// Mitsubishi GX Works2 project: IELET2103_Oving2   PLC: FX2N/FX2NC
// IELET2103_Oving2

// global labels: Global1
VAR_GLOBAL
  Nødstoppbryter : BOOL;
  Drasnor_inne : BOOL;
  Drasnor_ute : BOOL;
  Giver_for_port_oppe : BOOL;
  Giver_for_port_nede : BOOL;
  Kontaktor_for_opprulling : BOOL;
  Kontaktor_for_nedrrulling : BOOL;
  Lampe : BOOL;
END_VAR

// task Task_01 (event TRUE, interval 0, priority 31): Oppgave3

PROGRAM Oppgave1a)ST
VAR
  tmp1 : BOOL;
END_VAR
tmp1	:=	 X0 OR (NOT X1 AND M0) AND (M0<>X0) OR NOT M1;

M0 := tmp1; 
M1 :=	tmp1 AND X1;
END_PROGRAM

PROGRAM Oppgave1a)IL
// body in language c0 not rendered
END_PROGRAM

PROGRAM Oppgave1a)LD
(* structured ladder/FBD written out as ST: instructions are called as NAME(EN, inputs, outputs); _pN, _eN, _tN stand for wires *)
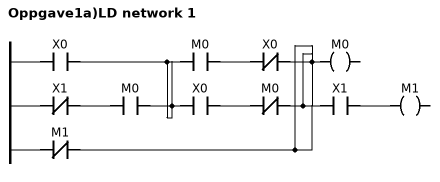
(* network 1 *)
_p1 := X0 OR (NOT X1 AND M0);
_p2 := (_p1 AND M0 AND NOT X0) OR (_p1 AND X0 AND NOT M0) OR (NOT M1);
M0 := _p2;
M1 := _p2 AND X1;
END_PROGRAM

PROGRAM Oppgave1b)LD
(* structured ladder/FBD written out as ST: instructions are called as NAME(EN, inputs, outputs); _pN, _eN, _tN stand for wires *)
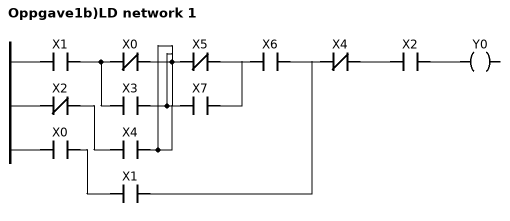
(* network 1 *)
_p1 := (X1 AND NOT X0) OR (X1 AND X3) OR (NOT X2 AND X4);
Y0 := (((((_p1 AND NOT X5) OR (_p1 AND X7)) AND X6) OR (X0 AND X1)) AND NOT X4) AND X2;
END_PROGRAM

PROGRAM Oppgave1b)ST
VAR
  block1 : BOOL;
  block2 : BOOL;
  block3 : BOOL;
  block4 : BOOL;
END_VAR
(*Oppgave 1b) ST*)

block1 := X1 AND (NOT X0 OR X3);
block2 := NOT X2 AND X4;
block3 := (block1 OR block2) AND (NOT X5 OR X7) AND X6;
block4 := block3 OR (X0 AND X1)
 
Y0 := block4 AND NOT X4 AND X2;
END_PROGRAM

PROGRAM Oppgave1c)
(* structured ladder/FBD written out as ST: instructions are called as NAME(EN, inputs, outputs); _pN, _eN, _tN stand for wires *)
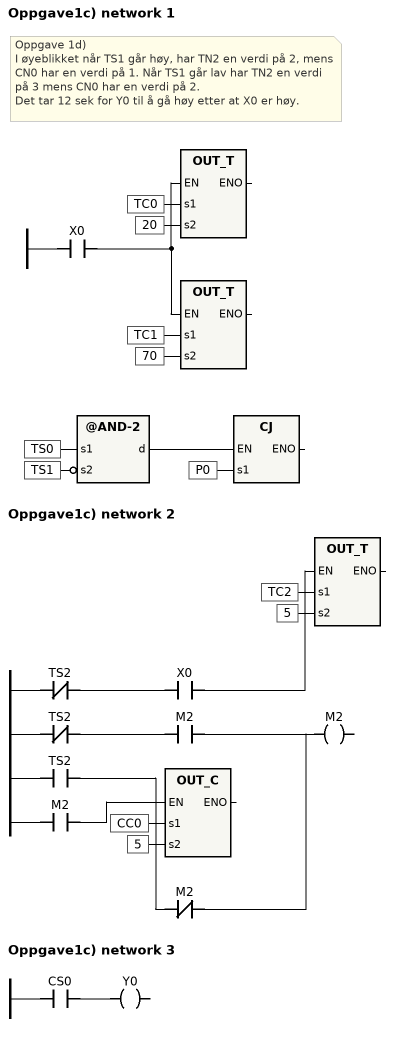
(* network 1 *)
(* Oppgave 1d)  / I øyeblikket når TS1 går høy, har TN2 en verdi på 2, mens CN0 har en verdi på 1. Når TS1 går lav har TN2 en verdi på 3 mens CN0 har en verdi på 2.   /  /  /  / Det tar 12 sek for Y0 til å gå høy etter at X0 er høy. *)
OUT_T(X0, TC0, 20);
OUT_T(X0, TC1, 70);
CJ(@AND-2(TS0, NOT TS1), P0);
(* network 2 *)
OUT_T(NOT TS2 AND X0, TC2, 5);
M2 := (NOT TS2 AND M2) OR (TS2 AND NOT M2);
OUT_C(M2, CC0, 5);
(* network 3 P0: *)
Y0 := CS0;
END_PROGRAM

PROGRAM Oppgave2
(* structured ladder/FBD written out as ST: instructions are called as NAME(EN, inputs, outputs); _pN, _eN, _tN stand for wires *)
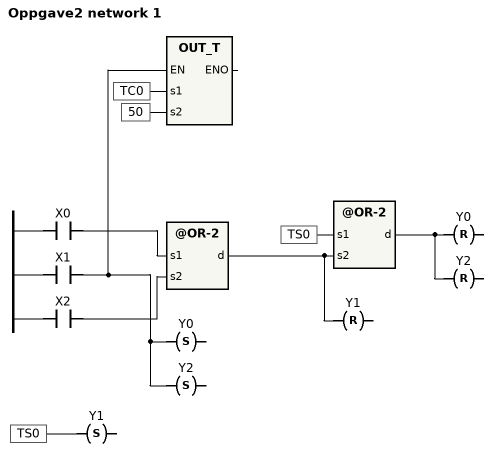
(* network 1 *)
SET(X1, Y0);
_p1 := @OR-2(X0, X2);
_p2 := @OR-2(TS0, _p1);
RST(_p2, Y0);
OUT_T(X1, TC0, 50);
SET(TS0, Y1);
RST(_p1, Y1);
SET(X1, Y2);
RST(_p2, Y2);
END_PROGRAM

PROGRAM Oppgave3
(* structured ladder/FBD written out as ST: instructions are called as NAME(EN, inputs, outputs); _pN, _eN, _tN stand for wires *)
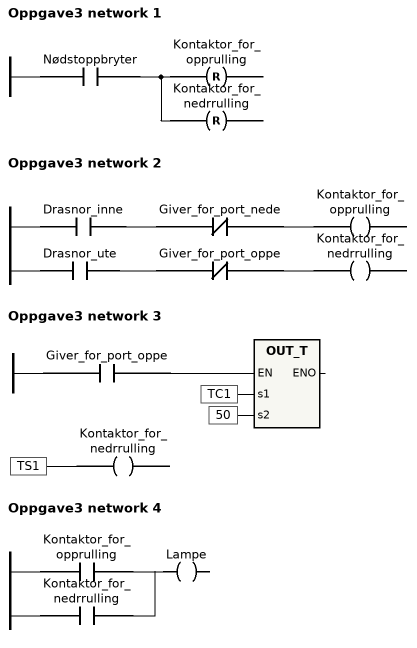
(* network 1 *)
RST(Nødstoppbryter, Kontaktor_for_opprulling);
RST(Nødstoppbryter, Kontaktor_for_nedrrulling);
(* network 2 *)
Kontaktor_for_opprulling := Drasnor_inne AND NOT Giver_for_port_nede;
Kontaktor_for_nedrrulling := Drasnor_ute AND NOT Giver_for_port_oppe;
(* network 3 *)
OUT_T(Giver_for_port_oppe, TC1, 50);
Kontaktor_for_nedrrulling := TS1;
(* network 4 *)
Lampe := Kontaktor_for_opprulling OR Kontaktor_for_nedrrulling;
END_PROGRAM
